# EPICS StreamDevice protocol: siteLibs/XGS600LibSrc/proto/XGS600.proto
# XGS-600 Stream protocol file

Terminator = CR;
ReplyTimeout = 1000;
ReadTimeout = 1000;

sw-ver-si {
    out "#\$105";
    in ">%s";
}

press1_si {
    out "#\$102UHFIG1";
    in ">%e";
    @mismatch {
        in ">%s";
    }
}
press2_si {
    out "#\$102UAUX1";
    in ">%e";
    @mismatch {
        in ">%s";
    }
}
press3_si {
    out "#\$102UAUX2";
    in ">%e";
    @mismatch {
        in ">%s";
    }
}
press4_si {
    out "#\$102UCNV1";
    in ">%e";
    @mismatch {
        in ">%s";
    }
}
press5_si {
    out "#\$102UCNV2";
    in ">%e";
    @mismatch {
        in ">%s";
    }
}

sys_reset {
    out "#\$106";
}

set_pres_unit {
    out "#\$11%d";
}

read_pres_unit {
    out "#\$113";
    in ">%d";
}

set_lock_on {
    out "#\$12%d";
}

read_lock_on {
    out "#\$122";
    in ">%d";
}

read_setpoint_st {
    out "#\$103";
    in ">00%x";
}

set_setpoint {
    out "#\$15E\$2%d";
}

read_setpoint {
    out "#\$15F%d";
    in ">%d";
}

set_setpoint_val {
    out "#\$16UHFIG111.000E-2";
}

set_setpoint_delay_on {
    out "#\$1C%d%.1f";
}

set_setpoint_delay_off {
    out "#\$1D%d%.1f";
}
